TYPE T_Ctrl_SIf_PRS_Cfg :
STRUCT
END_STRUCT
END_TYPE

(* stored: Version 1.1.0.1, ProductVersion 3.1.0.19
   DUT T_Ctrl_SIf_PRS_Cfg: Id {ab0eff3e-f125-40a6-9b44-b53f0ee42a0f} *)
